FUNCTION_BLOCK EL3681 EXTENDS EcSlaveInfoDataExt
VAR_INPUT
	MinValue												: 	LREAL 	:= 0.0;
	MaxValue												: 	LREAL 	:= 0.0;
	NoOfDigits												: 	INT 	(0..10)	:= 6; //number of decimal digits of scaled Q variable 
	OutOnError												:	LREAL 	:= 0.000000000000000001;
{attribute 'displaymode':='binary'}     	            	
	Options													:	BYTE  := 2#0000_0010; (* .0 = FALSE Scale value from 0 to e.g. 32767 / TRUE scale singed value e.g. -32768 <-> 32767 , see Options .1 and .2 for more scaling Options 
																						.1 = FALSE = 32 bit resolution / TRUE = value is based on 24 bit resolution e.g. -> -8388608.0 or 0.0 <-> 8388607.0 
																						.2 = Right adjust of 32/24 bit value -> value will be shifted by 8 bits (divided bv 256)   
																						.3 = TRUE = Enable extended range mode -> change scaling to +/-7812500 instead of r+/- 838860x *)
	Offset													:	LREAL := 0.0;
END_VAR                 									                                	            	
VAR_OUTPUT                              	            	
	Q														:	LREAL;	//scaled result value
{attribute 'displaymode':='binary'}     	            	
	Status										AT  %I*		:	WORD := 2#0100_0000_0000_0000;	//Terminal status word -> can also be linked with status byte

	In											AT  %I* 	: 	DINT; 	//Hardware Input 

	ActMode													: 	BYTE; //Setting Mode: 	0 = [V] DC | 1 = [V] AC 	| 2 = [A] DC 	| 3 = [A] AC
	ActRange												: 	BYTE; //Setting Range: 255 = 0.3 	| 1 = 3 		| 2 = 30 		| 3 = 300 

{attribute 'displaymode':='hex'}
	Control										AT%Q*		: 	WORD;   
    	
END_VAR
VAR	
{attribute 'displaymode':='hex'}
	Settings									AT  %I*		:	WORD; //Actual setting for mode and range 
END_VAR

SUPER^();

(* Scaling ******************************************************************)
	IF MaxValue <> MinValue 
	THEN
		IF Options.1 
		THEN //24 bit resolution
			IF NOT Options.3
			THEN
				Q 	 										:= Offset + Scale(SEL(Options.2 , In , In / 256.0 ) , SEL(Options.0, 0.0, -8388608.0), 8388607.0, MinValue , MaxValue);
			ELSE
		 		Q 	 										:= Offset + Scale(SEL(Options.2 , In , In / 256.0 ) , SEL(Options.0, 0.0, -7812500.0), 7812500.0, MinValue , MaxValue);
			END_IF
		ELSE //32 bit resolution 
			Q 	 											:= Offset + Scale(SEL(Options.2 , In , In / 256.0 ) , SEL(Options.0, 0.0, -2147483648.0), 2147483647.0, MinValue , MaxValue);		
		END_IF
		IF NoOfDigits > 0
		THEN
			Q												:= TO_FMLREAL(Q,NoOfDigits);
		END_IF
	
	ELSIF NoOfDigits > 0 (* Bsp PT100 *)
	THEN
		Q													:= Offset + TO_FMLREAL(In,NoOfDigits);
		
	ELSE  													
		Q 													:= 0.0;
	END_IF

	IF inError AND OutOnError <> 0.000000000000000001
	THEN
		Q													:= OutOnError;
	END_IF
	
(* Mode & Range **************************************************************)
	ActMode.0 												:= Settings.4;
	ActMode.1 												:= Settings.5;
	ActMode.2 												:= Settings.6;
	ActMode.3 												:= Settings.7;
	
	ActRange.0 												:= Settings.8;
	ActRange.1 												:= Settings.9;
	ActRange.2 												:= Settings.10;
	ActRange.3 												:= Settings.11;
	ActRange.4 												:= Settings.12;
    ActRange.5 												:= Settings.13;
    ActRange.6 												:= Settings.14;
    ActRange.7 												:= Settings.15;

(*****************************************************************************)

{attribute 'monitoring' := 'call'}
PROPERTY PUBLIC autorangeIsDisabled : BOOL
GET
autorangeIsDisabled := Status.5;
END_GET
END_PROPERTY

{attribute 'monitoring' := 'call'}
PROPERTY PUBLIC calibrationInProgress : BOOL
GET
calibrationInProgress := Status.7;
END_GET
END_PROPERTY

{attribute 'monitoring' := 'call'}
PROPERTY PUBLIC dataInvalid : BOOL
GET
dataInvalid := Status.3;
END_GET
END_PROPERTY

{attribute 'monitoring' := 'call'}
PROPERTY PUBLIC disableAutorange : BOOL
GET
DisableAutorange 	:= Control.0;
END_GET
SET
Control.0 								:= DisableAutorange;
END_SET
END_PROPERTY

{attribute 'monitoring' := 'call'}
PROPERTY PUBLIC inError : BOOL
GET
InError					:= Status.6 OR MinValue = MaxValue AND NoOfDigits = 0;
END_GET
END_PROPERTY

{attribute 'monitoring' := 'call'}
PROPERTY PUBLIC inExtendedRange : BOOL
GET
inExtendedRange := Status.2;
END_GET
END_PROPERTY

{attribute 'monitoring' := 'call'}
PROPERTY PUBLIC overrange : BOOL
GET
overrange 		:= status.1;
END_GET
END_PROPERTY

{attribute 'monitoring' := 'call'}
PROPERTY PUBLIC rangeInvalid : BOOL
GET
rangeInvalid := Status.4;
END_GET
END_PROPERTY

{attribute 'monitoring' := 'call'}
// 0 = [V] DC | 1 = [V] AC | 2 = [A] DC | 3 = [A] AC
PROPERTY PUBLIC setControlMode : INT
GET
setControlMode.0 := Control.4;
setControlMode.1 := Control.5;
setControlMode.2 := Control.6;
setControlMode.3 := Control.7;
END_GET
SET
Control.4 := setControlMode.0;
Control.5 := setControlMode.1;
Control.6 := setControlMode.2;
Control.7 := setControlMode.3;
END_SET
END_PROPERTY

{attribute 'monitoring' := 'call'}
// 	disable autorange to use range
// 	255 = 0.3 		| 1 = 3 		| 2 = 30 		| 3 = 300 
//	255 = 3*10^-1 	| 1 = 3*10^0 	| 2 = 3*10^1 	| 3 = 3*10^2 
PROPERTY PUBLIC setControlRange : INT
GET
setControlRange.0 := Control.8;
setControlRange.1 := Control.9;
setControlRange.2 := Control.10;
setControlRange.3 := Control.11;
setControlRange.4 := Control.12;
setControlRange.5 := Control.13;
setControlRange.6 := Control.14;
setControlRange.7 := Control.15;
END_GET
SET
Control.8 := setControlRange.0;
Control.9 := setControlRange.1;
Control.10 := setControlRange.2;
Control.11 := setControlRange.3;
Control.12 := setControlRange.4;
Control.13 := setControlRange.5;
Control.14 := setControlRange.6;
Control.15 := setControlRange.7;
END_SET
END_PROPERTY

{attribute 'monitoring' := 'call'}
PROPERTY PUBLIC startCalibration : BOOL
GET
StartCalibration 	:= Control.1;
END_GET
SET
Control.1 								:= StartCalibration;
END_SET
END_PROPERTY

{attribute 'monitoring' := 'call'}
PROPERTY PUBLIC underrange : BOOL
GET
underrange 		:= status.0;
END_GET
END_PROPERTY

END_FUNCTION_BLOCK

(* stored: Version 1.1.0.1, ProductVersion 3.1.4024.13
   POU EL3681: Id {8c2c280e-0811-4294-b658-b4042616ecd5}, SpecialFunc None
   Property autorangeIsDisabled: Id {6aac41de-6a14-4da5-8ec4-7cc807ffdb19}
   Get Get: Id {96c5cac8-449e-41e2-99a8-5b6612c407b6}
   Property calibrationInProgress: Id {118a5291-ec56-482d-acf7-59bb46d71142}
   Get Get: Id {067d7aec-ffb2-4fa7-a1be-5a0aec3b6530}
   Property dataInvalid: Id {4ed2eef0-80c5-4f79-ac33-191bf3263a35}
   Get Get: Id {b00533e6-7b7f-46fd-a331-93aca327bd82}
   Property disableAutorange: Id {43dbe815-4cd8-4ef0-890c-5458091aec81}
   Get Get: Id {1d76c3e0-1920-49be-89ce-0830479a805a}
   Set Set: Id {48fce614-8f30-45aa-8171-00183daa03d0}
   Property inError: Id {b877242c-0491-458f-b94d-14363ea67eec}
   Get Get: Id {8adb7e3a-3e76-4bef-a91f-8fcb6e5e197a}
   Property inExtendedRange: Id {3842ee38-b201-4aef-80ff-7b12d26fa15b}
   Get Get: Id {470350ab-ac68-4d51-b768-0b8125633e84}
   Property overrange: Id {c92ded85-77b9-406c-a4be-185651aab3db}
   Get Get: Id {58d636da-dec7-4cea-9e85-e4bb7e421043}
   Property rangeInvalid: Id {62d80656-c744-4731-b069-aa3c1b2c5a58}
   Get Get: Id {c772c669-a72b-44a0-9632-53296b562812}
   Property setControlMode: Id {4b29490d-6d7b-49e3-99a8-3b85f2dd9427}
   Get Get: Id {eab59895-0588-4dcc-b0b3-3b7e9e147361}
   Set Set: Id {8f532f7d-de2e-4d6b-a300-c05ef80f8859}
   Property setControlRange: Id {99d68934-98c4-404d-a682-fa7d9706ce7d}
   Get Get: Id {f9e5c2c4-3fbd-4475-9267-587f506f6056}
   Set Set: Id {2e2c3c4b-fb8c-4b19-8919-d0f6c43b22fc}
   Property startCalibration: Id {33d23d62-e588-4932-b3e4-aa0e3d6f7b68}
   Get Get: Id {debd7513-d0ca-4b94-ac91-755dacefcb1d}
   Set Set: Id {f1e9df9f-4482-4211-a5e1-94b4591ced85}
   Property underrange: Id {eda3de2a-af3d-4f07-a3c6-f41c11c87494}
   Get Get: Id {7fdaaf16-49a1-40ae-978b-f170cb40cc7e} *)
